{attribute 'conditionalshow'}
FUNCTION_BLOCK FB_CV_WORD_TO_BOOL
VAR_INPUT
	{attribute 'hide'}
	wInputValue			: WORD;								//Input value that is converted into the output value
END_VAR
VAR_OUTPUT
	{attribute 'hide'}
	arrOutputValue		: ARRAY[0..15] OF BOOL;				//Converted output value
END_VAR
VAR
END_VAR

//Creator : Kai Ebensperger
//Company : Lynus AG
//Date : 28.04.2021
//Version : 1.0.0.0

//With this functionblock its possible to convert a certain Datatyp in a other Datatype
//WORD TO BOOL
//Created for the Edge Device Lib over Modbus TCP
//Modbus TCP is WORD oriented

arrOutputValue[0] := wInputValue.0;
arrOutputValue[1] := wInputValue.1;
arrOutputValue[2] := wInputValue.2;
arrOutputValue[3] := wInputValue.3;
arrOutputValue[4] := wInputValue.4;
arrOutputValue[5] := wInputValue.5;
arrOutputValue[6] := wInputValue.6;
arrOutputValue[7] := wInputValue.7;
arrOutputValue[8] := wInputValue.8;
arrOutputValue[9] := wInputValue.9;
arrOutputValue[10] := wInputValue.10;
arrOutputValue[11] := wInputValue.11;
arrOutputValue[12] := wInputValue.12;
arrOutputValue[13] := wInputValue.13;
arrOutputValue[14] := wInputValue.14;
arrOutputValue[15] := wInputValue.15;

END_FUNCTION_BLOCK

(* stored: Version 1.1.0.1, ProductVersion 3.1.4024.9
   POU FB_CV_WORD_TO_BOOL: Id {cdffff38-0715-482f-b69b-5e93e95f4395}, SpecialFunc None *)
